# EPICS substitutions: db/Beckhoff_KL/ecmcC9900-M995.substitutions
file "ecmcEcSlave.template"
{
  pattern {}
          {}
}

file "ecmcC9900-M995-chx.template"
{
  pattern {CH_ID}
          {1    }
          {2    }
          {3    }
          {4    }
          {5    }
          {6    }
          {7    }
          {8    }
          {9    }
          {10   }
}
